FUNCTION_BLOCK FB_CTD_UDINT (* Down counter (UDINT) *)
  (* Standard: 61499-1; Description: Copyright (c) 2023 Martin Erich Jobst This program and the accompanying materials are made available under the terms of the Eclipse Public License 2.0 which is available at https://www.eclipse.org/legal/epl-2.0/ SPDX-License-Identifier: EPL-2.0 *)
  (* Version 3.0, 2025-04-14, Patrick Aigner, changed package *)
  (* Version 1.0, 2023-04-28, Martin Jobst *)
  PACKAGE iec61131::counters;
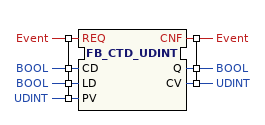
  EVENT_INPUT
    REQ WITH CD, PV, LD; (* Normal Execution Request *)
  END_EVENT
  EVENT_OUTPUT
    CNF WITH Q, CV; (* Execution Confirmation *)
  END_EVENT
  VAR_INPUT
    CD : BOOL; (* Count down *)
    LD : BOOL; (* Load *)
    PV : UDINT; (* Preset value *)
  END_VAR
  VAR_OUTPUT
    Q : BOOL; (* Output *)
    CV : UDINT; (* Count value *)
  END_VAR
  EC_STATES
    REQ : REQ -> CNF;
  END_STATES
  ALGORITHM REQ IN ST:
IF LD THEN
	CV := PV;
ELSIF CD AND CV > 0 THEN
	CV := CV - 1;
END_IF;
Q := CV <= 0;
  END_ALGORITHM
END_FUNCTION_BLOCK
